{attribute 'GeneratedUsingTerminal: EL3751-0000-0020'}
{attribute addProperty BoxType "EL3751-0000-0020"}
{attribute addProperty Id "StartTimeNextLatchAT %I*StartTimeNextLatch_02E0C1C88"}
{attribute addProperty CRC "1841615510"}
{attribute addProperty Size "8"}
TYPE PAI_Timestamp_6DC4D296 EXTENDS InputBase_8311D824 :
STRUCT
	{attribute addProperty Name "StartTimeNextLatch"}
	StartTimeNextLatch AT %I* : StartTimeNextLatch_02E0C1C8;
END_STRUCT
END_TYPE

(* stored: Version 1.2.0.0, ProductVersion 3.1.4024.9
   DUT PAI_Timestamp_6DC4D296: Id {5d7ac43f-14b1-4242-8501-86d3844d6bdb} *)
